(* PLC project coef_scale, Dassault Systèmes ControlBuild 2024x *)
(* stored: creationDateTime 2023-10-03T11:13:32-01:00 *)

(* This module simulates a scaling equation. Form of the scaling equation is y = k x . *)
FUNCTION_BLOCK equipment_library.coef_scale
  VAR_INPUT
    inputValue : REAL := 0.0;
  END_VAR
  VAR_OUTPUT
    outputValue : REAL := 0.0;
  END_VAR
  VAR CONSTANT
    coefficient : REAL := 1.0;
  END_VAR
  VAR
    d_scale : BOOL := false;
    v_d_scale : REAL := 0.0;
  END_VAR


ACTION C_source_code:
/* ----------------------------------------------------------------	*/
/* Type : Model of Operative Behaviour					*/
/* Category :  Toolbox							*/
/* Author : Dassault Systemes						*/
/* Update date : June 2018						*/
/* ----------------------------------------------------------------	*/
/* This module simulates the scaling of real variables			*/
/*	by multiplying it by a parameter coefficient.			*/
/* Form of the scaling equation is y = k x .				*/
/* ----------------------------------------------------------------	*/

if (d_scale)
	outputValue = v_d_scale;
else
	outputValue = inputValue * coefficient;
END_ACTION
END_FUNCTION_BLOCK
